// TIA Portal project "109482830_Target_1500S_PROJ_V12_V16" (V16)

(* hardware
DEVICE "PC-System_1"  CPU 1515SP PC
   slot 0: "PC-System_1"  CPU 1515SP PC F  6ES7 677-2WBx2-0xB0  V2.5
      slot 124: "Diagbase"  Diagbase  V6.0.4
      slot 125: "PC-System_1"  PC Station 2.3  Station_Manager  V2.3
   slot 1: "Software PLC_1"  CPU 1505SP TF  6ES7 672-5WC11-0YA0  V2.5
      slot 3: "CPU display_1"  6ES7591-1BA00-0AA0
   slot 2: "PROFINET onboard_2"  IE General  IE_CP  V2.2.0
   slot 127: "BA 2xRJ45"  BA 2xRJ45  6ES7 193-6AR00-0AA0  V0.0
      slot 32769: "Port_1"  6ES7 193-6AR00-0AA0
      slot 32770: "Port_2"  6ES7 193-6AR00-0AA0
   slot 1002: "Server module_1"  Server module  6ES7 193-6PA00-0AA0  V1.1
      slot 1: "Server module_1"  Server module
*)

// ===== PLC "Software PLC_1"  CPU 1505SP TF =====

TYPE "ModelPIDParams"
// This block is AUTO GENERATED - DO NOT MODIFY this block!
// Created by ODK_CodeGenerator version 205.0.2601.8
// at Tue April 30 14:11:13 2019
// ********************************************************
   STRUCT
      ModelPID_PIDController_D : LReal;   // [PIDController/D Gain/Internal Parameters/Derivative Gain]:ModelPID_P.PIDController_D
      ModelPID_PIDController_I : LReal;   // [PIDController/I Gain/Internal Parameters/Integral Gain]:ModelPID_P.PIDController_I
      ModelPID_PIDController_InitialConditionForFilter : LReal;   // [PIDController/Filter/Disc. Forward Euler Filter/Filter]:ModelPID_P.PIDController_InitialConditionForFilter
      ModelPID_PIDController_InitialConditionForIntegrator : LReal;   // [PIDController/Integrator/Discrete/Integrator]:ModelPID_P.PIDController_InitialConditionForIntegrator
      ModelPID_PIDController_LowerSaturationLimit : LReal;   // [PIDController/Saturation/Enabled/Saturation]:ModelPID_P.PIDController_LowerSaturationLimit
      ModelPID_PIDController_N : LReal;   // [PIDController/N Gain/Internal Parameters/Filter Coefficient]:ModelPID_P.PIDController_N
      ModelPID_PIDController_P : LReal;   // [PIDController/Parallel P Gain/Internal Parameters/Proportional Gain]:ModelPID_P.PIDController_P
      ModelPID_PIDController_UpperSaturationLimit : LReal;   // [PIDController/Saturation/Enabled/Saturation]:ModelPID_P.PIDController_UpperSaturationLimit
      ModelPID_Integrator_gainval : LReal;   // [PIDController/Integrator/Discrete/Integrator]:ModelPID_P.Integrator_gainval
      ModelPID_Filter_gainval : LReal;   // [PIDController/Filter/Disc. Forward Euler Filter/Filter]:ModelPID_P.Filter_gainval
      ModelPID_Gain_Gain : LReal;   // [Gain]:ModelPID_P.Gain_Gain
      ModelPID_Gain1_Gain : LReal;   // [Gain1]:ModelPID_P.Gain1_Gain
   END_STRUCT;
END_TYPE

TYPE "ModelPIDExtModeStatus"
// This PLC data type is used to show the status of internal functions called in ModelPIDCallExtMode FB.
   STRUCT
      Status_TCON : Word;   // This is the status of TCON block called in ModelPIDCallExtMode FB. Please refer to the STEP 7 documentation of TCON block for possible values of this parameter.
      Status_TDISCON : Word;   // This is the status of TDISCON block called in ModelPIDCallExtMode FB. Please refer to the STEP 7 documentation of TDISCON block for possible values of this parameter.
      Status_TRCV : Word;   // This is the status of TRCV block called in ModelPIDCallExtMode FB. Please refer to the STEP 7 documentation of TRCV block for possible values of this parameter.
      Status_TSEND : Word;   // This is the status of TSEND block called in ModelPIDCallExtMode FB. Please refer to the STEP 7 documentation of TSEND block for possible values of this parameter.
      Status_ODK : Int;   // This is the status of ModelPIDExtModeInternal ODK 1500S FB which is called in ModelPIDCallExtMode FB. Please refer to the ODK 1500S documentation for possible values of this parameter.
      Status_ExtMode : Word;   // This is the status code for Target 1500S specific error cases. Please refer to the Target 1500S documentation for possible values of this parameter.
   END_STRUCT;
END_TYPE

TYPE "ModelPIDInternalModelSignals"
// This block is AUTO GENERATED - DO NOT MODIFY this block!
// Created by ODK_CodeGenerator version 205.0.2601.8
// at Tue April 30 14:11:13 2019
// ********************************************************
   STRUCT
      sig_sum : LReal;
      outpid : LReal;
      setpoint : LReal;
      processval : LReal;
   END_STRUCT;
END_TYPE

DATA_BLOCK "GlobalParameters"   // DB1
{ S7_Optimized_Access := 'TRUE' }
VERSION : 0.1
   VAR
      setpoint : LReal;
      process : LReal;
      outPID : LReal;
      statusOneStep : Word;
      statusExternalMode : "ModelPIDExtModeStatus";
      paramAccess : Bool := true;
      writeActive : Bool;
      parameters : "ModelPIDParams";
      statusParameters : Word;
      internalSignals : "ModelPIDInternalModelSignals";
      statusUnload : Word;
      statusLoad : Word;
   END_VAR
BEGIN
   statusExternalMode.Status_TCON := 16#7002;
   statusExternalMode.Status_TDISCON := 16#0000;
   statusExternalMode.Status_TRCV := 16#0000;
   statusExternalMode.Status_TSEND := 16#0000;
   statusExternalMode.Status_ODK := 0;
   statusExternalMode.Status_ExtMode := 16#0000;
END_DATA_BLOCK

// folder: 01_Startup

DATA_BLOCK "InstModelPID_Unload"   // DB2
{ S7_Optimized_Access := 'TRUE' }
VERSION : 0.1
// stored: InstanceOfName ModelPID_Unload
"ModelPID_Unload"
BEGIN
END_DATA_BLOCK

DATA_BLOCK "InstModelPID_Load"   // DB3
{ S7_Optimized_Access := 'TRUE' }
VERSION : 0.1
// stored: InstanceOfName ModelPID_Load
"ModelPID_Load"
BEGIN
END_DATA_BLOCK

// folder: 02_Cyclic/01_ProcessAndPID

DATA_BLOCK "InstLSim_PT3"   // DB4
{ S7_Optimized_Access := 'TRUE' }
VERSION : 2.0
// stored: InstanceOfName LSim_PT3
"LSim_PT3"
BEGIN
END_DATA_BLOCK

DATA_BLOCK "InstModelPIDOneStep"   // DB5
{ S7_Optimized_Access := 'TRUE' }
VERSION : 0.1
// stored: InstanceOfName ModelPIDOneStep
"ModelPIDOneStep"
BEGIN
END_DATA_BLOCK

// folder: 02_Cyclic/02_ExternalMode

DATA_BLOCK "InstModelPIDCallExtMode"   // DB6
{ S7_Optimized_Access := 'TRUE' }
VERSION : 0.1
// stored: InstanceOfName ModelPIDCallExtMode
"ModelPIDCallExtMode"
BEGIN
END_DATA_BLOCK

// folder: 02_Cyclic/03_ReadWriteParameters

DATA_BLOCK "InstModelPIDReadWriteParameters"   // DB7
{ S7_Optimized_Access := 'TRUE' }
VERSION : 0.1
// stored: InstanceOfName ModelPIDReadWriteParameters
"ModelPIDReadWriteParameters"
BEGIN
END_DATA_BLOCK

// folder: 02_Cyclic/04_WebReadWrite

DATA_BLOCK "gDB_SWV_Interface"   // DB8
{ S7_Optimized_Access := 'TRUE' }
VERSION : 0.1
// stored: InstanceOfName ModelPIDWebReadWrite
"ModelPIDWebReadWrite"
BEGIN
END_DATA_BLOCK

// folder: 01_Startup

FUNCTION_BLOCK "ModelPID_Load"   // FB1, SCL
{ S7_Optimized_Access := 'TRUE' }
VERSION : 0.1
// This block is AUTO GENERATED - DO NOT MODIFY this block!
// Created by ODK_CodeGenerator version 205.0.2601.8
// at Tue April 30 14:11:13 2019
// max. number of parallel calls into this ODK application is: 1
// *************************************************************
   VAR_INPUT
      REQ : Bool;
   END_VAR
   VAR_OUTPUT
      DONE : Bool;
      BUSY : Bool;
      ERROR : Bool;
      STATUS : Int;
   END_VAR
   VAR
      ODK_Load_Instance : ODK_Load;
      _odk_internal_LIBRARY_NAME : String := '<rt>ModelPID_ODK.so';
   END_VAR
   VAR CONSTANT
      _odk_internal_INSTANCE_ID : UDInt := 1_489_625_180;
   END_VAR
BEGIN
   //
   // DO NOT CHANGE BELOW OF THIS LINE !!
   // This is an automatic generated block by the
   // SIMATIC ODK 1500S V2.5
   // DO NOT CHANGE !!
   //
   #ODK_Load_Instance(REQ := #REQ,
                      LIBRARY_NAME := #_odk_internal_LIBRARY_NAME,
                      INSTANCE_ID := #_odk_internal_INSTANCE_ID,
                      DONE => #DONE,
                      BUSY => #BUSY,
                      ERROR => #ERROR,
                      STATUS => #STATUS);
   //
   // DO NOT CHANGE !!
   // This is an automatic generated block by the
   // SIMATIC ODK 1500S V2.5
   // DO NOT CHANGE ABOVE OF THIS LINE !!
   //
END_FUNCTION_BLOCK

FUNCTION_BLOCK "ModelPID_Unload"   // FB2, SCL
{ S7_Optimized_Access := 'TRUE' }
VERSION : 0.1
// This block is AUTO GENERATED - DO NOT MODIFY this block!
// Created by ODK_CodeGenerator version 205.0.2601.8
// at Tue April 30 14:11:13 2019
// max. number of parallel calls into this ODK application is: 1
// *************************************************************
   VAR_INPUT
      REQ : Bool;
   END_VAR
   VAR_OUTPUT
      DONE : Bool;
      BUSY : Bool;
      ERROR : Bool;
      STATUS : Int;
   END_VAR
   VAR
      ODK_Unld_Instance : ODK_Unld;
   END_VAR
   VAR CONSTANT
      _odk_internal_INSTANCE_ID : UDInt := 1_489_625_180;
   END_VAR
BEGIN
   //
   // DO NOT CHANGE BELOW OF THIS LINE !!
   // This is an automatic generated block by the
   // SIMATIC ODK 1500S V2.5
   // DO NOT CHANGE !!
   //
   #ODK_Unld_Instance(REQ := #REQ,
                      INSTANCE_ID := #_odk_internal_INSTANCE_ID,
                      DONE => #DONE,
                      BUSY => #BUSY,
                      ERROR => #ERROR,
                      STATUS => #STATUS);
   //
   // DO NOT CHANGE !!
   // This is an automatic generated block by the
   // SIMATIC ODK 1500S V2.5
   // DO NOT CHANGE ABOVE OF THIS LINE !!
   //
END_FUNCTION_BLOCK

ORGANIZATION_BLOCK "Startup"   // OB100, LAD, Startup
TITLE = "Complete Restart"
{ S7_Optimized_Access := 'TRUE' }
VERSION : 0.1
   VAR_INPUT
      LostRetentive : Bool;   // True if retentive data are lost
      LostRTC : Bool;   // True if date and time are lost
   END_VAR
BEGIN

REGION Network 1: Unload current SO-File
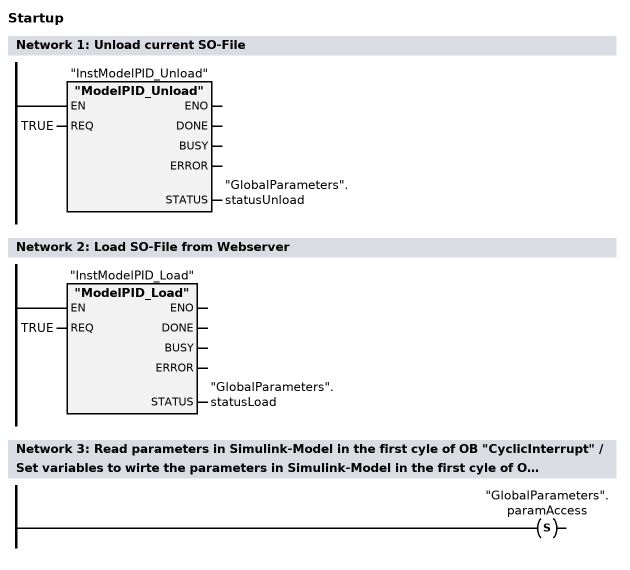
   RUNG wire#powerrail
      "InstModelPID_Unload"(REQ := TRUE, DONE =>, BUSY =>, ERROR =>, STATUS => "GlobalParameters".statusUnload)
   END_RUNG
   // the same network as SCL:
   "InstModelPID_Unload"(REQ := TRUE, STATUS => "GlobalParameters".statusUnload);   // "ModelPID_Unload"
END_REGION

REGION Network 2: Load SO-File from Webserver
   RUNG wire#powerrail
      "InstModelPID_Load"(REQ := TRUE, DONE =>, BUSY =>, ERROR =>, STATUS => "GlobalParameters".statusLoad)
   END_RUNG
   // the same network as SCL:
   "InstModelPID_Load"(REQ := TRUE, STATUS => "GlobalParameters".statusLoad);   // "ModelPID_Load"
END_REGION

REGION Network 3: Read parameters in Simulink-Model in the first cyle of OB "CyclicInterrupt" / Set variables to wirte the parameters in Simulink-Model in the first cyle of OB "CyclicInterrupt"
   RUNG wire#powerrail
      S_Coil( "GlobalParameters".paramAccess )
   END_RUNG
   // the same network as SCL:
   "GlobalParameters".paramAccess := TRUE;
END_REGION
END_ORGANIZATION_BLOCK

// folder: 02_Cyclic

ORGANIZATION_BLOCK "CyclicInterrupt"   // OB30, LAD, CyclicInterrupt
TITLE = Cycle 100 ms
{ S7_Optimized_Access := 'TRUE' }
VERSION : 0.1
   VAR_INPUT
      Initial_Call : Bool;   // Initial call of this OB
      Event_Count : Int;   // Events discarded
   END_VAR
   VAR_TEMP   // added for the SCL form of the ladder/FBD networks
      _w1 : Bool;
   END_VAR
BEGIN

REGION Network 1: Call simulation block for temperature process
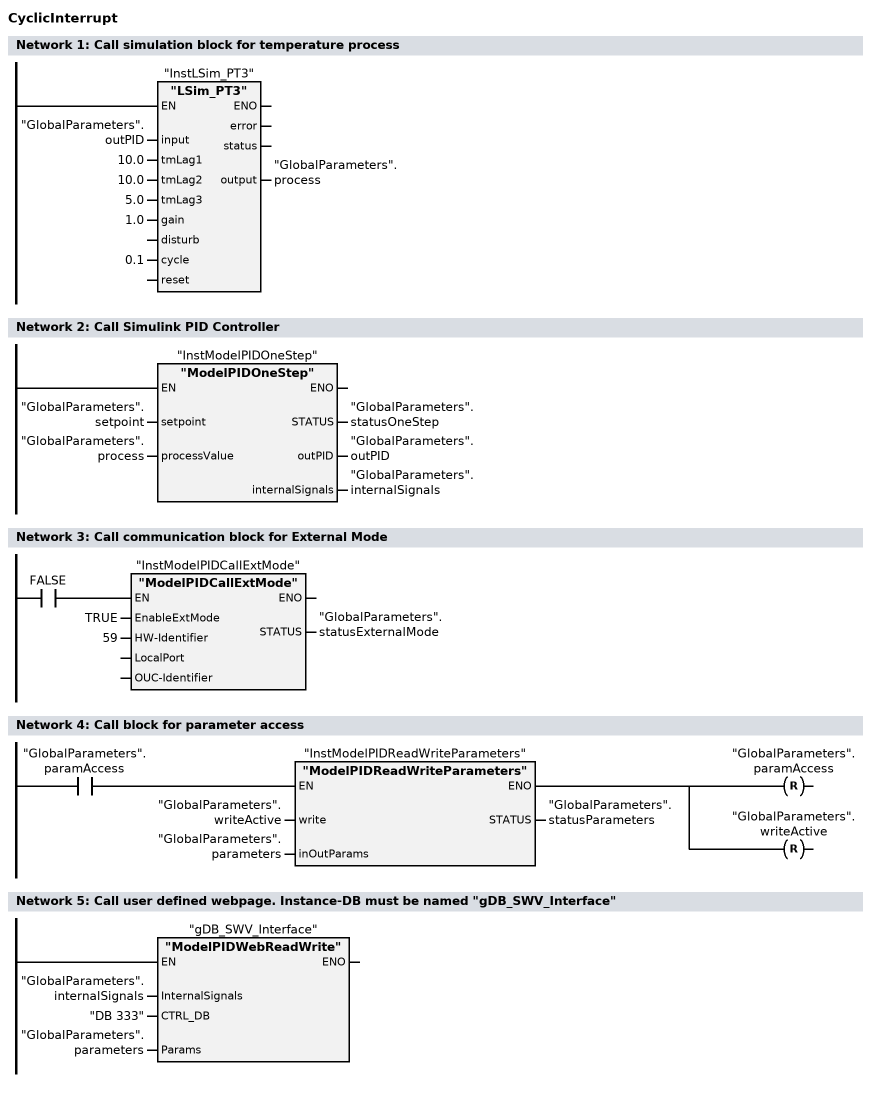
   RUNG wire#powerrail
      "InstLSim_PT3"(input := "GlobalParameters".outPID, tmLag1 := 10.0, tmLag2 := 10.0, tmLag3 := 5.0, gain := 1.0, disturb :=, cycle := 0.1, reset :=, error =>, status =>, output => "GlobalParameters".process)
   END_RUNG
   // the same network as SCL:
   "InstLSim_PT3"(input := "GlobalParameters".outPID,   // "LSim_PT3"
                  tmLag1 := 10.0,
                  tmLag2 := 10.0,
                  tmLag3 := 5.0,
                  gain := 1.0,
                  cycle := 0.1,
                  output => "GlobalParameters".process);
END_REGION

REGION Network 2: Call Simulink PID Controller
   RUNG wire#powerrail
      "InstModelPIDOneStep"(setpoint := "GlobalParameters".setpoint, processValue := "GlobalParameters".process, STATUS => "GlobalParameters".statusOneStep, outPID => "GlobalParameters".outPID, internalSignals => "GlobalParameters".internalSignals)
   END_RUNG
   // the same network as SCL:
   "InstModelPIDOneStep"(setpoint := "GlobalParameters".setpoint,   // "ModelPIDOneStep"
                         processValue := "GlobalParameters".process,
                         STATUS => "GlobalParameters".statusOneStep,
                         outPID => "GlobalParameters".outPID,
                         internalSignals => "GlobalParameters".internalSignals);
END_REGION

REGION Network 3: Call communication block for External Mode
   RUNG wire#powerrail
      Contact( FALSE )
      "InstModelPIDCallExtMode"(EnableExtMode := TRUE, "HW-Identifier" := 59, LocalPort :=, "OUC-Identifier" :=, STATUS => "GlobalParameters".statusExternalMode)
   END_RUNG
   // the same network as SCL:
   IF FALSE THEN
       "InstModelPIDCallExtMode"(EnableExtMode := TRUE,   // "ModelPIDCallExtMode"
                               "HW-Identifier" := 59,
                               STATUS => "GlobalParameters".statusExternalMode);
   END_IF;
END_REGION

REGION Network 4: Call block for parameter access
   RUNG wire#powerrail
      Contact( "GlobalParameters".paramAccess )
      "InstModelPIDReadWriteParameters"(write := "GlobalParameters".writeActive, inOutParams := "GlobalParameters".parameters, STATUS => "GlobalParameters".statusParameters)
      wire#w1
      R_Coil( "GlobalParameters".paramAccess )
   END_RUNG
   RUNG wire#w1
      R_Coil( "GlobalParameters".writeActive )
   END_RUNG
   // the same network as SCL:
   "InstModelPIDReadWriteParameters"(EN := "GlobalParameters".paramAccess,   // "ModelPIDReadWriteParameters"
                           write := "GlobalParameters".writeActive,
                           inOutParams := "GlobalParameters".parameters,
                           STATUS => "GlobalParameters".statusParameters,
                           ENO => #_w1);
   IF #_w1 THEN
       "GlobalParameters".paramAccess := FALSE;
       "GlobalParameters".writeActive := FALSE;
   END_IF;
END_REGION

REGION Network 5: Call user defined webpage. Instance-DB must be named "gDB_SWV_Interface"
   RUNG wire#powerrail
      "gDB_SWV_Interface"(InternalSignals := "GlobalParameters".internalSignals, CTRL_DB := "DB 333", Params := "GlobalParameters".parameters)
   END_RUNG
   // the same network as SCL:
   "gDB_SWV_Interface"(InternalSignals := "GlobalParameters".internalSignals,   // "ModelPIDWebReadWrite"
                       CTRL_DB := "DB 333",
                       Params := "GlobalParameters".parameters);
END_REGION
END_ORGANIZATION_BLOCK

// folder: 02_Cyclic/01_ProcessAndPID

FUNCTION_BLOCK "ModelPIDOneStep"   // FB3, SCL
{ S7_Optimized_Access := 'TRUE' }
VERSION : 0.1
// This block is AUTO GENERATED - DO NOT MODIFY this block!
// Created by ODK_CodeGenerator version 205.0.2601.8
// at Tue April 30 14:11:13 2019
// max. number of parallel calls into this ODK application is: 1
// *************************************************************
//  This is generated by Target 1500S for Simulink
//  Model name:                  ModelPID
//  Model version:               1.149
//                 
//  ODK 1500S version:           V2.5
//  Target 1500S version:        V3.0         
//  MATLAB version:              9.5 (R2018b) 24-May-2018
//  Simulink version:            9.2 (R2018b) 24-May-2018
//  MATLAB Coder version:        4.1 (R2018b) 24-May-2018
//  Simulink Coder version:      9.0 (R2018b) 24-May-2018
//  
//  ***Model details***
//  Step Size:                   0.1
//  Default parameter behaviour: Tunable
//  External Mode:               On
//  Allow OneStep and
//  CallExtMode FBs to be
//  called in different OBs      No
//  
//  ***ODK 1500S details***  
//  Heap Size:                   32k
//  Max Block Size:              1024
//  Size of thread stack:        32k
//  SyncCallParallelCount:       1(max. number of parallel calls into this ODK application)
//  ********************************************************
   VAR_INPUT
      setpoint : LReal;
      processValue : LReal;
   END_VAR
   VAR_OUTPUT
      STATUS : Int := 0;
      outPID : LReal;
      internalSignals : "ModelPIDInternalModelSignals";
   END_VAR
   VAR
      _odk_internal_Last_REQ : Bool := FALSE;
      _odk_internal_Last_BUSY : Bool := FALSE;
      _odk_internal_IN_BUFFER : Array[0..15] of Byte;
      _odk_internal_OUT_BUFFER : Array[0..39] of Byte;
   END_VAR
   VAR_TEMP
      _odk_internal_pos : DInt;
      _odk_internal_err : Int;
      _odk_internal_i : DInt;
   END_VAR
   VAR CONSTANT
      _odk_internal_INSTANCE_ID : UDInt := 1_489_625_180;
      _odk_internal_COMMAND : UDInt := 1_728_603_471;
   END_VAR
BEGIN
   //
   // DO NOT CHANGE BELOW OF THIS LINE !!
   // This is an automatic generated block by the
   // SIMATIC ODK 1500S V2.5
   // DO NOT CHANGE !!
   //
   // This is generated by Target 1500S for Simulink
   // Model name:                  ModelPID
   // Model version:               1.149
   //                
   // ODK 1500S version:           V2.5
   // Target 1500S version:        V3.0         
   // MATLAB version:              9.5 (R2018b) 24-May-2018
   // Simulink version:            9.2 (R2018b) 24-May-2018
   // MATLAB Coder version:        4.1 (R2018b) 24-May-2018
   // Simulink Coder version:      9.0 (R2018b) 24-May-2018
   // 
   // ***Model details***
   // Step Size:                   0.1
   // Default parameter behaviour: Tunable
   // External Mode:               On
   // Allow OneStep and
   // CallExtMode FBs to be
   // called in different OBs      No
   // 
   // ***ODK 1500S details***  
   // Heap Size:                   32k
   // Max Block Size:              1024
   // Size of thread stack:        32k
   // SyncCallParallelCount:       1(max. number of parallel calls into this ODK application)
   // ********************************************************
   // 
   #_odk_internal_pos := 0;
   #_odk_internal_err := WRITE_LITTLE(src_variable := #setpoint, dest_array := #_odk_internal_IN_BUFFER, pos := #_odk_internal_pos);
   #_odk_internal_err := WRITE_LITTLE(src_variable := #processValue, dest_array := #_odk_internal_IN_BUFFER, pos := #_odk_internal_pos);
   #STATUS := ODK_ExcS(INSTANCE_ID := #_odk_internal_INSTANCE_ID,
                       COMMAND := #_odk_internal_COMMAND,
                       IN_DATA := #_odk_internal_IN_BUFFER,
                       INOUT_DATA := null,
                       OUT_DATA := #_odk_internal_OUT_BUFFER
   );
   IF INT_TO_UINT(#STATUS) < 16#7000 THEN
       #_odk_internal_pos := 0;
       #_odk_internal_err := READ_LITTLE(dest_Variable => #outPID, src_array := #_odk_internal_OUT_BUFFER, pos := #_odk_internal_pos);
       #_odk_internal_err := READ_LITTLE(dest_Variable => #internalSignals.#sig_sum, src_array := #_odk_internal_OUT_BUFFER, pos := #_odk_internal_pos);
       #_odk_internal_err := READ_LITTLE(dest_Variable => #internalSignals.#outpid, src_array := #_odk_internal_OUT_BUFFER, pos := #_odk_internal_pos);
       #_odk_internal_err := READ_LITTLE(dest_Variable => #internalSignals.#setpoint, src_array := #_odk_internal_OUT_BUFFER, pos := #_odk_internal_pos);
       #_odk_internal_err := READ_LITTLE(dest_Variable => #internalSignals.#processval, src_array := #_odk_internal_OUT_BUFFER, pos := #_odk_internal_pos);
   END_IF;
   //
   // DO NOT CHANGE !!
   // This is an automatic generated block by the
   // SIMATIC ODK 1500S V2.5
   // DO NOT CHANGE ABOVE OF THIS LINE !!
   //
END_FUNCTION_BLOCK

FUNCTION_BLOCK "LSim_PT3"   // FB54, SCL
{ S7_Optimized_Access := 'TRUE' }
VERSION : 2.0
   VAR_INPUT
      input : Real;   // input variable
      tmLag1 : Real := 29.0;   // time lag 1 in s
      tmLag2 : Real := 17.5;   // time lag 2 in s
      tmLag3 : Real := 3.1;   // time lag 3 in s
      gain : Real := 1.0;   // proportional gain
      disturb : Real;   // disturbance variable (additional to "input")
      cycle : Real := 0.1;   // sample time [in sec]
      reset : Bool;   // complete restart (#output = #input)
   END_VAR
   VAR_OUTPUT
      error : Bool;   // error (#tmLag1 <= 0 or #tmLag2 <= 0 or #tmLag3 <= 0)
      status : Word;   // status (if #error = TRUE then status = 16#8001)
      output : Real;   // output signal (if #error = FALSE)
   END_VAR
   VAR
      statFback1 : Real;   // feedback path value 1
      statFback2 : Real;   // feedback path value 2
      statFback3 : Real;   // feedback path value 3
   END_VAR
   VAR_TEMP
      tempHvar : Real;   // help variable
      tempCycleR : Real;   // cycle to real
      tempTmLag1R : Real;   // time lag 1 to real
      tempTmLag2R : Real;   // time lag 2 to real
      tempTmLag3R : Real;   // time lag 3 to real
      tempOutvNew : Real;   // new output variable
   END_VAR
BEGIN
   //=============================================================================
   //SIEMENS AG
   //(c)Copyright 2016 All Rights Reserved
   //-----------------------------------------------------------------------------
   //Library:       Library for Controlled System Simulation
   //Tested with:   S7-1500 FW V1.8
   //Engineering:   STEP 7 Prof. V13 SP1 Upd6 (TIA Portal)
   //Restrictions:  Cyclic interrupt
   //Requirements:  memory card needed
   //Functionality: Simulation of an PT3-system
   //
   //                               gain
   //  F(p) = ------------------------------------------------------
   //         (tmLag1 * p + 1) * (tmLag2 * p + 1) * (tmLag3 * p + 1)
   //          
   //  Call the simulation in a cyclic interrupt with
   //  cyclic interrupt time at least = tmLag1/10!
   //-----------------------------------------------------------------------------
   //Change log table:
   //Version  Date       Expert in charge                Changes applied
   //02.00.00 03.02.2016 Siemens Industry Online Support Release (STEP 7 V13 SP1)
   //=============================================================================

   // check parameter
   IF #tmLag1 <= 0 OR #tmLag2 <= 0 OR #tmLag3 <= 0 THEN
     #error := TRUE;
     #status := W#16#8001;     // Parameter Error
     #output := #input; //write output data
     #statFback1 := #input; //write static data
     #statFback2 := #input;
     #statFback3 := #input;
     RETURN;
   ELSE
     #error := FALSE;
     #status := W#16#0000;     // no error
   END_IF;

   IF #reset THEN //complete restart routine

     #output := #input;//write output data
     #statFback1 := #input;//write static data
     #statFback2 := #input;
     #statFback3 := #input;

   ELSE //cycle mode routine

     #tempCycleR  := #cycle*1000; //transform data type
     #tempTmLag1R := #tmLag1*1000;
     #tempTmLag2R := #tmLag2*1000;
     #tempTmLag3R := #tmLag3*1000;

     IF #tempCycleR * 0.5 > #tempTmLag1R THEN //limit TM_LAG1
       #tempTmLag1R := #tempCycleR * 0.5;
     END_IF;

     IF #tempCycleR * 0.5 > #tempTmLag2R THEN //limit TM_LAG2
       #tempTmLag2R := #tempCycleR * 0.5;
     END_IF;

     IF #tempCycleR * 0.5 > #tempTmLag3R THEN //limit TM_LAG2
       #tempTmLag3R := #tempCycleR * 0.5;
     END_IF;

     //1. first order lag algorithm
     #tempHvar     := #tempCycleR / (#tempTmLag1R * 2.0); 
     #tempHvar     := (#gain * (#input + #disturb) - #statFback1) * #tempHvar / (#tempHvar + 1.0);
     #tempOutvNew  := #tempHvar + #statFback1;
     #statFback1  := #tempHvar * 2.0 + #statFback1;

     //2. first order lag algorithm
     #tempHvar     := #tempCycleR / (#tempTmLag2R * 2.0); 
     #tempHvar     := ((#tempOutvNew - #statFback2) * #tempHvar) / (#tempHvar + 1.0);
     #tempOutvNew  := #tempHvar + #statFback2;
     #statFback2  := #tempHvar * 2.0 + #statFback2;

     //3. first order lag algorithm
     #tempHvar     := #tempCycleR / (#tempTmLag3R * 2.0); 
     #tempHvar     := ((#tempOutvNew - #statFback3) * #tempHvar) / (#tempHvar + 1.0);
     #tempOutvNew  := #tempHvar + #statFback3;
     #statFback3  := #tempHvar * 2.0 + #statFback3;

     #output := #tempOutvNew; //write output

   END_IF;
END_FUNCTION_BLOCK

// folder: 02_Cyclic/02_ExternalMode

FUNCTION_BLOCK "ModelPIDExtModeInternal"   // FB4, SCL
{ S7_Optimized_Access := 'TRUE' }
VERSION : 0.1
// This block is AUTO GENERATED - DO NOT MODIFY this block!
// Created by ODK_CodeGenerator version 205.0.2601.8
// at Tue April 30 14:11:13 2019
// max. number of parallel calls into this ODK application is: 1
// *************************************************************
//  This is generated by Target 1500S for Simulink
//  Model name:                  ModelPID
//  Model version:               1.149
//                 
//  ODK 1500S version:           V2.5
//  Target 1500S version:        V3.0         
//  MATLAB version:              9.5 (R2018b) 24-May-2018
//  Simulink version:            9.2 (R2018b) 24-May-2018
//  MATLAB Coder version:        4.1 (R2018b) 24-May-2018
//  Simulink Coder version:      9.0 (R2018b) 24-May-2018
//  
//  ***Model details***
//  Step Size:                   0.1
//  Default parameter behaviour: Tunable
//  External Mode:               On
//  Allow OneStep and
//  CallExtMode FBs to be
//  called in different OBs      No
//  
//  ***ODK 1500S details***  
//  Heap Size:                   32k
//  Max Block Size:              1024
//  Size of thread stack:        32k
//  SyncCallParallelCount:       1(max. number of parallel calls into this ODK application)
//  ********************************************************
//  
//  This function will be used internally for External Mode. Please do not call this function
   VAR_INPUT
      receiveLength : UDInt;
      stateIn : UDInt;
   END_VAR
   VAR_OUTPUT
      STATUS : Int := 0;
      sendLength : UDInt;
      funcError : Bool;
      funcStatus : Word;
      stateOut : UDInt;
   END_VAR
   VAR_IN_OUT
      bufferToModel : Array[0..65535] of Byte;
      bufferFromModel : Array[0..65535] of Byte;
   END_VAR
   VAR
      _odk_internal_Last_REQ : Bool := FALSE;
      _odk_internal_Last_BUSY : Bool := FALSE;
      _odk_internal_IN_BUFFER : Array[0..7] of Byte;
      _odk_internal_INOUT_BUFFER : Array[0..131071] of Byte;
      _odk_internal_OUT_BUFFER : Array[0..10] of Byte;
   END_VAR
   VAR_TEMP
      _odk_internal_pos : DInt;
      _odk_internal_err : Int;
      _odk_internal_i : DInt;
   END_VAR
   VAR CONSTANT
      _odk_internal_INSTANCE_ID : UDInt := 1_489_625_180;
      _odk_internal_COMMAND : UDInt := 940_238_321;
   END_VAR
BEGIN
   //
   // DO NOT CHANGE BELOW OF THIS LINE !!
   // This is an automatic generated block by the
   // SIMATIC ODK 1500S V2.5
   // DO NOT CHANGE !!
   //
   // This is generated by Target 1500S for Simulink
   // Model name:                  ModelPID
   // Model version:               1.149
   //                
   // ODK 1500S version:           V2.5
   // Target 1500S version:        V3.0         
   // MATLAB version:              9.5 (R2018b) 24-May-2018
   // Simulink version:            9.2 (R2018b) 24-May-2018
   // MATLAB Coder version:        4.1 (R2018b) 24-May-2018
   // Simulink Coder version:      9.0 (R2018b) 24-May-2018
   // 
   // ***Model details***
   // Step Size:                   0.1
   // Default parameter behaviour: Tunable
   // External Mode:               On
   // Allow OneStep and
   // CallExtMode FBs to be
   // called in different OBs      No
   // 
   // ***ODK 1500S details***  
   // Heap Size:                   32k
   // Max Block Size:              1024
   // Size of thread stack:        32k
   // SyncCallParallelCount:       1(max. number of parallel calls into this ODK application)
   // ********************************************************
   // 
   // This function will be used internally for External Mode. Please do not call this function
   #_odk_internal_pos := 0;
   #_odk_internal_err := WRITE_LITTLE(src_variable := #receiveLength, dest_array := #_odk_internal_IN_BUFFER, pos := #_odk_internal_pos);
   #_odk_internal_err := WRITE_LITTLE(src_variable := #stateIn, dest_array := #_odk_internal_IN_BUFFER, pos := #_odk_internal_pos);
   #_odk_internal_pos := 0;
   MOVE_BLK(COUNT := 65536,
            IN := #bufferToModel[0],
            OUT => #_odk_internal_INOUT_BUFFER[#_odk_internal_pos]);
   #_odk_internal_pos := #_odk_internal_pos + 65536;
   MOVE_BLK(COUNT := 65536,
            IN := #bufferFromModel[0],
            OUT => #_odk_internal_INOUT_BUFFER[#_odk_internal_pos]);
   #_odk_internal_pos := #_odk_internal_pos + 65536;
   #STATUS := ODK_ExcS(INSTANCE_ID := #_odk_internal_INSTANCE_ID,
                       COMMAND := #_odk_internal_COMMAND,
                       IN_DATA := #_odk_internal_IN_BUFFER,
                       INOUT_DATA := #_odk_internal_INOUT_BUFFER,
                       OUT_DATA := #_odk_internal_OUT_BUFFER
   );
   IF INT_TO_UINT(#STATUS) < 16#7000 THEN
       #_odk_internal_pos := 0;
       MOVE_BLK(COUNT := 65536,
                IN := #_odk_internal_INOUT_BUFFER[#_odk_internal_pos],
                OUT => #bufferToModel[0]);
       #_odk_internal_pos := #_odk_internal_pos + 65536;
       MOVE_BLK(COUNT := 65536,
                IN := #_odk_internal_INOUT_BUFFER[#_odk_internal_pos],
                OUT => #bufferFromModel[0]);
       #_odk_internal_pos := #_odk_internal_pos + 65536;
       #_odk_internal_pos := 0;
       #_odk_internal_err := READ_LITTLE(dest_Variable => #sendLength, src_array := #_odk_internal_OUT_BUFFER, pos := #_odk_internal_pos);
       #funcError := BYTE_TO_BOOL(#_odk_internal_OUT_BUFFER[#_odk_internal_pos]);
       #_odk_internal_pos := #_odk_internal_pos + 1;
       #_odk_internal_err := READ_LITTLE(dest_Variable => #funcStatus, src_array := #_odk_internal_OUT_BUFFER, pos := #_odk_internal_pos);
       #_odk_internal_err := READ_LITTLE(dest_Variable => #stateOut, src_array := #_odk_internal_OUT_BUFFER, pos := #_odk_internal_pos);
   END_IF;
   //
   // DO NOT CHANGE !!
   // This is an automatic generated block by the
   // SIMATIC ODK 1500S V2.5
   // DO NOT CHANGE ABOVE OF THIS LINE !!
   //
END_FUNCTION_BLOCK

FUNCTION_BLOCK "ModelPIDCallExtMode"   // FB6, SCL
{ S7_Optimized_Access := 'TRUE' }
VERSION : 0.1
// This block is AUTO GENERATED - DO NOT MODIFY this block!
// Created by Target 1500S version V3.0
// at 2019-04-30 14:10:49 
// ********************************************************
//  This is generated by Target 1500S for Simulink
//  Model name:                  ModelPID
//  Model version:               1.149
//                
//  ODK 1500S version:           V2.5
//  Target 1500S version:        V3.0         
//  MATLAB version:              9.5 (R2018b) 24-May-2018
//  Simulink version:            9.2 (R2018b) 24-May-2018
//  MATLAB Coder version:        4.1 (R2018b) 24-May-2018
//  Simulink Coder version:      9.0 (R2018b) 24-May-2018
// 
//  ***Model details***
//  Step Size:                   0.1
//  Default parameter behaviour: Tunable 
//  External Mode:               On
//  Allow OneStep and
//  CallExtMode FBs to be
//  called in different OBs      No
// 
//  ***ODK 1500S details***  
//  Heap Size:                   32k
//  Max Block Size:              1024
//  Size of thread stack:        32k
//  SyncCallParallelCount:       1(max. number of parallel calls into this ODK application)
//  ********************************************************
// Call this FB to establish a connection to Simulink PC for External Mode.
   VAR_INPUT
      EnableExtMode : Bool;
      "HW-Identifier" : UInt := 59;
      LocalPort : UInt := 17725;
      "OUC-Identifier" : Conn_Ouc := 1;
   END_VAR
   VAR_OUTPUT
      STATUS : "ModelPIDExtModeStatus";
   END_VAR
   VAR
      TCON_Instance : TCON;
      TDISCON_Instance : TDISCON;
      TRCV_Instance : TRCV;
      TSEND_Instance : TSEND;
      ModelPIDExtMode_Instance : "ModelPIDExtModeInternal";
      tconParam : TCON_IP_v4;
      tconREQ : Bool;
      tconDONE : Bool;
      tconBUSY : Bool;
      tconERROR : Bool;
      tdisconREQ : Bool;
      tdisconDONE : Bool;
      tdisconERROR : Bool;
      tdisconBUSY : Bool;
      trcvDONE : Bool;
      trcvERROR : Bool;
      trcvBUSY : Bool;
      trcvRCVD_LEN : UDInt;
      tsendREQ : Bool;
      tsendDONE : Bool;
      tsendBUSY : Bool;
      tsendERROR : Bool;
      tsendGrcREQ : Bool;
      tsendGrcDONE : Bool;
      tsendGrcBUSY : Bool;
      tsendGrcERROR : Bool;
      tsendGrcSTATUS : Word;
      extModeOdkStatus : Int;
      extModeFuncStatus : Word;
      extModeFuncError : Bool;
      extModeRCVD_LEN : UDInt;
      st_STATUS : "ModelPIDExtModeStatus";
      prev_state : UDInt;
      state : UDInt := 0;
      messageBuf : Array[1..8] of Byte;
      dataExchangeBufToModel : Array[1..#BUF_SIZE] of Byte;
      dataExchangeBufFromModel : Array[1..#BUF_SIZE] of Byte;
   END_VAR
   VAR CONSTANT
      BUF_SIZE : UDInt := 65536;   // 64k
      ST_IDLE : UDInt := 0;
      ST_RECEIVE : UDInt := 1;
      ST_SEND : UDInt := 2;
      ST_DISCON : UDInt := 3;
      ST_DISCON_GRACEFULL : UDInt := 4;
      ST_EXEC_ODK : UDInt := 5;
      EXT_MODEL_SHUTDOWN : Byte := 16#14;
   END_VAR
BEGIN
   // This is generated by Target 1500S for Simulink
   // Model name:                  ModelPID
   // Model version:               1.149
   //               
   // ODK 1500S version:           V2.5
   // Target 1500S version:        V3.0         
   // MATLAB version:              9.5 (R2018b) 24-May-2018
   // Simulink version:            9.2 (R2018b) 24-May-2018
   // MATLAB Coder version:        4.1 (R2018b) 24-May-2018
   // Simulink Coder version:      9.0 (R2018b) 24-May-2018
   //
   // ***Model details***
   // Step Size:                   0.1
   // Default parameter behaviour: Tunable 
   // External Mode:               On
   // Allow OneStep and
   // CallExtMode FBs to be
   // called in different OBs      No
   //
   // ***ODK 1500S details***  
   // Heap Size:                   32k
   // Max Block Size:              1024
   // Size of thread stack:        32k
   // SyncCallParallelCount:       1(max. number of parallel calls into this ODK application)
   // ********************************************************
   //Call this FB to establish a connection to Simulink PC for External Mode.

   IF NOT #EnableExtMode THEN
       RETURN;
   END_IF;
   #tconParam.ID := #"OUC-Identifier";
   #tconParam.LocalPort := #"LocalPort";
   #tconParam.InterfaceId := #"HW-Identifier";

   IF #state <> #ST_EXEC_ODK THEN
       #prev_state := #state;
   END_IF;

   CASE #state OF
       #ST_IDLE:
           IF NOT #tconBUSY THEN
               #tconREQ := NOT #tconREQ;
           END_IF;
           #TCON_Instance(REQ := #tconREQ,
                          ID := #tconParam.ID,
                          DONE => #tconDONE,
                          BUSY => #tconBUSY,
                          ERROR => #tconERROR,
                          STATUS => #st_STATUS.Status_TCON,
                          CONNECT := #tconParam);
           IF #tconDONE THEN
               #state := #ST_RECEIVE;
           END_IF;
       #ST_RECEIVE:
           #TRCV_Instance(EN_R := TRUE,
                          ID := #tconParam.ID,
                          LEN := #BUF_SIZE,
                          ADHOC := TRUE,
                          NDR => #trcvDONE,
                          BUSY => #trcvBUSY,
                          ERROR => #trcvERROR,
                          STATUS => #st_STATUS.Status_TRCV,
                          RCVD_LEN => #trcvRCVD_LEN,
                          DATA := #dataExchangeBufToModel);
           #state := #ST_EXEC_ODK;
       #ST_SEND:
           IF NOT #tsendBUSY THEN
               #tsendREQ := NOT #tsendREQ;
           END_IF;
           #TSEND_Instance(REQ := #tsendREQ,
                           ID := #tconParam.ID,
                           LEN := #extModeRCVD_LEN,
                           DONE => #tsendDONE,
                           BUSY => #tsendBUSY,
                           ERROR => #tsendERROR,
                           STATUS => #st_STATUS.Status_TSEND,
                           DATA := #dataExchangeBufFromModel);

           IF #tsendDONE THEN
               #state := #ST_RECEIVE;
           ELSIF #tsendERROR THEN
               #state := #ST_DISCON;
           ELSE
               #state := #ST_EXEC_ODK;
           END_IF;
       #ST_EXEC_ODK:
           #ModelPIDExtMode_Instance(stateIn := #prev_state,
                                     stateOut => #state,
                                     receiveLength := #trcvRCVD_LEN,
                                     sendLength => #extModeRCVD_LEN,
                                     STATUS => #st_STATUS.Status_ODK,
                                     funcError => #extModeFuncError,
                                     funcStatus => #st_STATUS.Status_ExtMode,
                                     bufferToModel := #dataExchangeBufToModel,
                                     bufferFromModel := #dataExchangeBufFromModel);
           IF #st_STATUS.Status_ODK <> 0 THEN
               #state := #ST_DISCON_GRACEFULL;
           END_IF;
       #ST_DISCON:
           IF NOT #tdisconBUSY THEN
               #tdisconREQ := NOT #tdisconREQ;
           END_IF;
           #extModeRCVD_LEN := 0;
           #trcvRCVD_LEN := 0;
           #TDISCON_Instance(REQ := #tdisconREQ,
                             ID := #tconParam.ID,
                             DONE => #tdisconDONE,
                             BUSY => #tdisconBUSY,
                             ERROR => #tdisconERROR,
                             STATUS => #st_STATUS.Status_TDISCON);
           IF #tdisconDONE OR #tdisconERROR THEN
               #state := #ST_IDLE;
           END_IF;
       #ST_DISCON_GRACEFULL:
           IF NOT #tsendGrcBUSY THEN
               #tsendGrcREQ := NOT #tsendGrcREQ;
           END_IF;
           #messageBuf[1] := #EXT_MODEL_SHUTDOWN;
           #TSEND_Instance(REQ := #tsendGrcREQ,
                           ID := #tconParam.ID,
                           LEN := 8,
                           DONE => #tsendGrcDONE,
                           BUSY => #tsendGrcBUSY,
                           ERROR => #tsendGrcERROR,
                           DATA := #messageBuf);

           IF #tsendGrcDONE OR #tsendGrcERROR THEN
               #state := #ST_DISCON;
           END_IF;
   END_CASE;

   #STATUS.Status_TCON := #st_STATUS.Status_TCON;
   #STATUS.Status_TDISCON := #st_STATUS.Status_TDISCON;
   #STATUS.Status_TSEND := #st_STATUS.Status_TSEND;
   #STATUS.Status_TRCV := #st_STATUS.Status_TRCV;
   #STATUS.Status_ODK := #st_STATUS.Status_ODK;
   #STATUS.Status_ExtMode := #st_STATUS.Status_ExtMode;
END_FUNCTION_BLOCK

// folder: 02_Cyclic/03_ReadWriteParameters

FUNCTION_BLOCK "ModelPIDReadWriteParameters"   // FB5, SCL
{ S7_Optimized_Access := 'TRUE' }
VERSION : 0.1
// This block is AUTO GENERATED - DO NOT MODIFY this block!
// Created by ODK_CodeGenerator version 205.0.2601.8
// at Tue April 30 14:11:13 2019
// max. number of parallel calls into this ODK application is: 1
// *************************************************************
//  This is generated by Target 1500S for Simulink
//  Model name:                  ModelPID
//  Model version:               1.149
//                 
//  ODK 1500S version:           V2.5
//  Target 1500S version:        V3.0         
//  MATLAB version:              9.5 (R2018b) 24-May-2018
//  Simulink version:            9.2 (R2018b) 24-May-2018
//  MATLAB Coder version:        4.1 (R2018b) 24-May-2018
//  Simulink Coder version:      9.0 (R2018b) 24-May-2018
//  
//  ***Model details***
//  Step Size:                   0.1
//  Default parameter behaviour: Tunable
//  External Mode:               On
//  Allow OneStep and
//  CallExtMode FBs to be
//  called in different OBs      No
//  
//  ***ODK 1500S details***  
//  Heap Size:                   32k
//  Max Block Size:              1024
//  Size of thread stack:        32k
//  SyncCallParallelCount:       1(max. number of parallel calls into this ODK application)
//  ********************************************************
//  
//  Call this function to read or write parameters from/to Simulink Model.
//  Set write[IN] parameter to TRUE in order to write and set FALSE to read parameters
   VAR_INPUT
      write : Bool;
   END_VAR
   VAR_OUTPUT
      STATUS : Int := 0;
   END_VAR
   VAR_IN_OUT
      inOutParams : "ModelPIDParams";
   END_VAR
   VAR
      _odk_internal_Last_REQ : Bool := FALSE;
      _odk_internal_Last_BUSY : Bool := FALSE;
      _odk_internal_IN_BUFFER : Array[0..0] of Byte;
      _odk_internal_INOUT_BUFFER : Array[0..95] of Byte;
   END_VAR
   VAR_TEMP
      _odk_internal_pos : DInt;
      _odk_internal_err : Int;
      _odk_internal_i : DInt;
   END_VAR
   VAR CONSTANT
      _odk_internal_INSTANCE_ID : UDInt := 1_489_625_180;
      _odk_internal_COMMAND : UDInt := 2_137_970_399;
   END_VAR
BEGIN
   //
   // DO NOT CHANGE BELOW OF THIS LINE !!
   // This is an automatic generated block by the
   // SIMATIC ODK 1500S V2.5
   // DO NOT CHANGE !!
   //
   // This is generated by Target 1500S for Simulink
   // Model name:                  ModelPID
   // Model version:               1.149
   //                
   // ODK 1500S version:           V2.5
   // Target 1500S version:        V3.0         
   // MATLAB version:              9.5 (R2018b) 24-May-2018
   // Simulink version:            9.2 (R2018b) 24-May-2018
   // MATLAB Coder version:        4.1 (R2018b) 24-May-2018
   // Simulink Coder version:      9.0 (R2018b) 24-May-2018
   // 
   // ***Model details***
   // Step Size:                   0.1
   // Default parameter behaviour: Tunable
   // External Mode:               On
   // Allow OneStep and
   // CallExtMode FBs to be
   // called in different OBs      No
   // 
   // ***ODK 1500S details***  
   // Heap Size:                   32k
   // Max Block Size:              1024
   // Size of thread stack:        32k
   // SyncCallParallelCount:       1(max. number of parallel calls into this ODK application)
   // ********************************************************
   // 
   // Call this function to read or write parameters from/to Simulink Model.
   // Set write[IN] parameter to TRUE in order to write and set FALSE to read parameters
   #_odk_internal_pos := 0;
   IF (True = #write) THEN
       #_odk_internal_IN_BUFFER[#_odk_internal_pos] := BYTE#1;
   ELSE
       #_odk_internal_IN_BUFFER[#_odk_internal_pos] := BYTE#0;
   END_IF;
   #_odk_internal_pos := #_odk_internal_pos + 1;
   #_odk_internal_pos := 0;
   #_odk_internal_err := WRITE_LITTLE(src_variable := #inOutParams.#ModelPID_PIDController_D, dest_array := #_odk_internal_INOUT_BUFFER, pos := #_odk_internal_pos);
   #_odk_internal_err := WRITE_LITTLE(src_variable := #inOutParams.#ModelPID_PIDController_I, dest_array := #_odk_internal_INOUT_BUFFER, pos := #_odk_internal_pos);
   #_odk_internal_err := WRITE_LITTLE(src_variable := #inOutParams.#ModelPID_PIDController_InitialConditionForFilter, dest_array := #_odk_internal_INOUT_BUFFER, pos := #_odk_internal_pos);
   #_odk_internal_err := WRITE_LITTLE(src_variable := #inOutParams.#ModelPID_PIDController_InitialConditionForIntegrator, dest_array := #_odk_internal_INOUT_BUFFER, pos := #_odk_internal_pos);
   #_odk_internal_err := WRITE_LITTLE(src_variable := #inOutParams.#ModelPID_PIDController_LowerSaturationLimit, dest_array := #_odk_internal_INOUT_BUFFER, pos := #_odk_internal_pos);
   #_odk_internal_err := WRITE_LITTLE(src_variable := #inOutParams.#ModelPID_PIDController_N, dest_array := #_odk_internal_INOUT_BUFFER, pos := #_odk_internal_pos);
   #_odk_internal_err := WRITE_LITTLE(src_variable := #inOutParams.#ModelPID_PIDController_P, dest_array := #_odk_internal_INOUT_BUFFER, pos := #_odk_internal_pos);
   #_odk_internal_err := WRITE_LITTLE(src_variable := #inOutParams.#ModelPID_PIDController_UpperSaturationLimit, dest_array := #_odk_internal_INOUT_BUFFER, pos := #_odk_internal_pos);
   #_odk_internal_err := WRITE_LITTLE(src_variable := #inOutParams.#ModelPID_Integrator_gainval, dest_array := #_odk_internal_INOUT_BUFFER, pos := #_odk_internal_pos);
   #_odk_internal_err := WRITE_LITTLE(src_variable := #inOutParams.#ModelPID_Filter_gainval, dest_array := #_odk_internal_INOUT_BUFFER, pos := #_odk_internal_pos);
   #_odk_internal_err := WRITE_LITTLE(src_variable := #inOutParams.#ModelPID_Gain_Gain, dest_array := #_odk_internal_INOUT_BUFFER, pos := #_odk_internal_pos);
   #_odk_internal_err := WRITE_LITTLE(src_variable := #inOutParams.#ModelPID_Gain1_Gain, dest_array := #_odk_internal_INOUT_BUFFER, pos := #_odk_internal_pos);
   #STATUS := ODK_ExcS(INSTANCE_ID := #_odk_internal_INSTANCE_ID,
                       COMMAND := #_odk_internal_COMMAND,
                       IN_DATA := #_odk_internal_IN_BUFFER,
                       INOUT_DATA := #_odk_internal_INOUT_BUFFER,
                       OUT_DATA := null);
   IF INT_TO_UINT(#STATUS) < 16#7000 THEN
       #_odk_internal_pos := 0;
       #_odk_internal_err := READ_LITTLE(dest_Variable => #inOutParams.#ModelPID_PIDController_D, src_array := #_odk_internal_INOUT_BUFFER, pos := #_odk_internal_pos);
       #_odk_internal_err := READ_LITTLE(dest_Variable => #inOutParams.#ModelPID_PIDController_I, src_array := #_odk_internal_INOUT_BUFFER, pos := #_odk_internal_pos);
       #_odk_internal_err := READ_LITTLE(dest_Variable => #inOutParams.#ModelPID_PIDController_InitialConditionForFilter, src_array := #_odk_internal_INOUT_BUFFER, pos := #_odk_internal_pos);
       #_odk_internal_err := READ_LITTLE(dest_Variable => #inOutParams.#ModelPID_PIDController_InitialConditionForIntegrator, src_array := #_odk_internal_INOUT_BUFFER, pos := #_odk_internal_pos);
       #_odk_internal_err := READ_LITTLE(dest_Variable => #inOutParams.#ModelPID_PIDController_LowerSaturationLimit, src_array := #_odk_internal_INOUT_BUFFER, pos := #_odk_internal_pos);
       #_odk_internal_err := READ_LITTLE(dest_Variable => #inOutParams.#ModelPID_PIDController_N, src_array := #_odk_internal_INOUT_BUFFER, pos := #_odk_internal_pos);
       #_odk_internal_err := READ_LITTLE(dest_Variable => #inOutParams.#ModelPID_PIDController_P, src_array := #_odk_internal_INOUT_BUFFER, pos := #_odk_internal_pos);
       #_odk_internal_err := READ_LITTLE(dest_Variable => #inOutParams.#ModelPID_PIDController_UpperSaturationLimit, src_array := #_odk_internal_INOUT_BUFFER, pos := #_odk_internal_pos);
       #_odk_internal_err := READ_LITTLE(dest_Variable => #inOutParams.#ModelPID_Integrator_gainval, src_array := #_odk_internal_INOUT_BUFFER, pos := #_odk_internal_pos);
       #_odk_internal_err := READ_LITTLE(dest_Variable => #inOutParams.#ModelPID_Filter_gainval, src_array := #_odk_internal_INOUT_BUFFER, pos := #_odk_internal_pos);
       #_odk_internal_err := READ_LITTLE(dest_Variable => #inOutParams.#ModelPID_Gain_Gain, src_array := #_odk_internal_INOUT_BUFFER, pos := #_odk_internal_pos);
       #_odk_internal_err := READ_LITTLE(dest_Variable => #inOutParams.#ModelPID_Gain1_Gain, src_array := #_odk_internal_INOUT_BUFFER, pos := #_odk_internal_pos);
   END_IF;
   //
   // DO NOT CHANGE !!
   // This is an automatic generated block by the
   // SIMATIC ODK 1500S V2.5
   // DO NOT CHANGE ABOVE OF THIS LINE !!
   //
END_FUNCTION_BLOCK

// folder: 02_Cyclic/04_WebReadWrite

FUNCTION_BLOCK "ModelPIDWebReadWrite"   // FB7, SCL
{ S7_Optimized_Access := 'TRUE' }
VERSION : 0.1
// This block is AUTO GENERATED - DO NOT MODIFY this block!
// Created by Target 1500S version 0
// at 0 
// ********************************************************
//  This is generated by Target 1500S for Simulink
//  Model name:                  ModelPID
//  Model version:               1.149
//                
//  ODK 1500S version:           V2.5
//  Target 1500S version:        V3.0         
//  MATLAB version:              9.5 (R2018b) 24-May-2018
//  Simulink version:            9.2 (R2018b) 24-May-2018
//  MATLAB Coder version:        4.1 (R2018b) 24-May-2018
//  Simulink Coder version:      9.0 (R2018b) 24-May-2018
// 
//  ***Model details***
//  Step Size:                   0.1
//  Default parameter behaviour: Tunable 
//  External Mode:               On
//  Allow OneStep and
//  CallExtMode FBs to be
//  called in different OBs      No
// 
//  ***ODK 1500S details***  
//  Heap Size:                   32k
//  Max Block Size:              1024
//  Size of thread stack:        32k
//  SyncCallParallelCount:       1(max. number of parallel calls into this ODK application)
//  ********************************************************
// Call this FB to establish a connection to user defined Web page.
   VAR_INPUT
      InternalSignals : "ModelPIDInternalModelSignals";
      CTRL_DB : DB_WWW;
   END_VAR
   VAR_IN_OUT
      Params : "ModelPIDParams";
   END_VAR
   VAR
      TestPointedSignals : "ModelPIDInternalModelSignals";
      Parameter : "ModelPIDParams";
      RWParams_Instance : "ModelPIDReadWriteParameters";
      Write : Int := 0;
      RunTime : LReal;
   END_VAR
   VAR_TEMP
      ret : Int;
   END_VAR
BEGIN
   // This is generated by Target 1500S for Simulink
   // Model name:                  ModelPID
   // Model version:               1.149
   //               
   // ODK 1500S version:           V2.5
   // Target 1500S version:        V3.0         
   // MATLAB version:              9.5 (R2018b) 24-May-2018
   // Simulink version:            9.2 (R2018b) 24-May-2018
   // MATLAB Coder version:        4.1 (R2018b) 24-May-2018
   // Simulink Coder version:      9.0 (R2018b) 24-May-2018
   //
   // ***Model details***
   // Step Size:                   0.1
   // Default parameter behaviour: Tunable 
   // External Mode:               On
   // Allow OneStep and
   // CallExtMode FBs to be
   // called in different OBs      No
   //
   // ***ODK 1500S details***  
   // Heap Size:                   32k
   // Max Block Size:              1024
   // Size of thread stack:        32k
   // SyncCallParallelCount:       1(max. number of parallel calls into this ODK application)
   // ********************************************************
   //Call this FB to establish a connection to user defined Web page.
   #RunTime := #RunTime + 100.0;

   #TestPointedSignals := #InternalSignals;
   CASE #Write OF
       0:
           #RWParams_Instance(write := FALSE,
                              STATUS => #RWParams_Instance.STATUS,
                              inOutParams := #Parameter);
           #Params := #Parameter;
       1:
           // Wait for parameter be updated by the Web action
           ;
       2:
           #RWParams_Instance(write := TRUE,
                              STATUS => #RWParams_Instance.STATUS,
                              inOutParams := #Parameter);
           #Params := #Parameter;
           #Write := 0;
       ELSE
           // Not possible to reach
           ;
   END_CASE;

   #ret := WWW(#CTRL_DB);
END_FUNCTION_BLOCK